Universal Robots PolyScope program: straight floor demo.urp

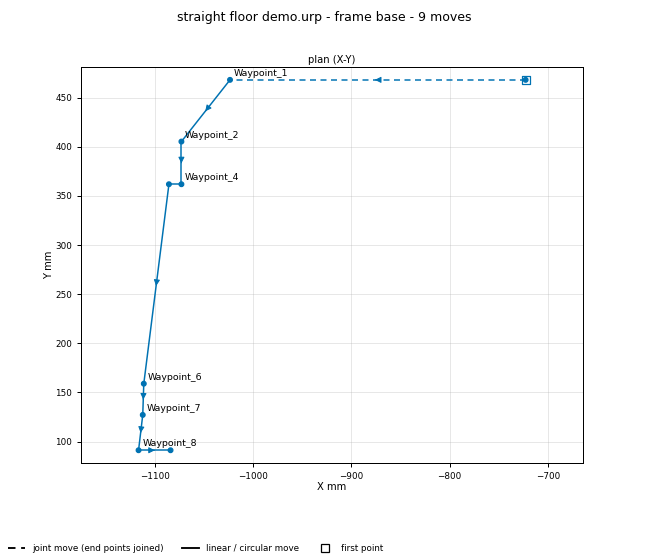
[picture p0: tool path of straight floor demo.urp in frame base, 9 of 9 moves have a stored position in this frame; points joined in program order, loops and branches not executed]
Program straight floor demo (installation=default directory=/programs createdIn=5.21.3 lastSavedIn=5.21.3 robotSerialNumber=20246801938)
Calibrated DH parameters: a=[-0.000071, -0.790281, -0.600694, 0.000061, -0.000039, 0]; d=[0.236272, 604.465945, 132.116513, -736.382239, 0.159268, 0.154005]; alpha=[1.570254, -0.000567, 0.000559, 1.571709, -1.56999, 0]; deltaTheta=[0, -0.409357, 7.293326, -0.600784, -0.000001, -0.000001]
InitVariablesNode
Robot Program (runOnlyOnce=false)
  Folder Folder1
    SuppressedNode
      MoveJ speed 60 deg/s, acceleration 80 deg/s^2 (useActiveTCP=true optimoveEnabled=false optiMoveSpeed=0.3 optiMoveAcceleration=0.09) feature=Base
        Waypoint oldhome: TCP in base x=397.354 y=356.263 z=319.809 mm, rx=2.3163 ry=2.0576 rz=0.0741 rad; joints [-198.308, -118.162, 133.452, -12.561, -11.517, -6.326] deg; TCP offset x=-9.5 y=-328 z=105.73 mm, rx=1.2092 ry=-1.2092 rz=1.2092 rad
    MoveJ speed 60 deg/s, acceleration 80 deg/s^2 (useActiveTCP=true optimoveEnabled=false optiMoveSpeed=0.3 optiMoveAcceleration=0.09) feature=Base
      Waypoint Waypoint_3: TCP in base x=-722.694 y=468.114 z=-58.679 mm, rx=-2.1116 ry=0.3311 rz=2.0412 rad; joints [-64.053, -54.316, 154.48, -187.789, -90.798, 312.597] deg
      Waypoint Waypoint_1: TCP in base x=-1023.509 y=468.114 z=-58.679 mm, rx=-2.1116 ry=0.3311 rz=2.0412 rad; joints [-42.99, -54.355, 134.192, -167.351, -89.902, 333.647] deg
    MoveL speed 20 mm/s, acceleration 1200 mm/s^2 (useActiveTCP=true optimoveEnabled=false optiMoveSpeed=0.3 optiMoveAcceleration=0.09) feature=Base
      Waypoint Waypoint_2: TCP in base x=-1072.965 y=405.321 z=-50.994 mm, rx=2.2388 ry=0.0055 rz=-2.1569 rad; joints [-42.937, -53.961, 129.721, -163.349, -90.663, 315.614] deg
      Waypoint Waypoint_4: TCP in base x=-1072.965 y=361.906 z=-50.994 mm, rx=2.2388 ry=0.0055 rz=-2.1569 rad; joints [-40.714, -54.402, 131.441, -164.605, -90.572, 317.835] deg
      Waypoint Waypoint_5: TCP in base x=-1085.671 y=361.906 z=-50.994 mm, rx=-2.2075 ry=0.1584 rz=2.13 rad; joints [-37.594, -54.591, 132.165, -165.084, -90.081, 329.433] deg
      Waypoint Waypoint_6: TCP in base x=-1111.256 y=158.94 z=-50.994 mm, rx=-2.2075 ry=0.1584 rz=2.13 rad; joints [-24.094, -55.21, 134.996, -167.356, -89.511, 342.92] deg
      Waypoint Waypoint_7: TCP in base x=-1112.305 y=127.176 z=-50.994 mm, rx=2.2506 ry=-0.0217 rz=-2.1687 rad; joints [-24.593, -55.191, 134.842, -167.171, -89.831, 335.324] deg
      Waypoint Waypoint_8: TCP in base x=-1116.578 y=91.213 z=-50.994 mm, rx=2.2506 ry=-0.0217 rz=-2.1687 rad; joints [-22.045, -55.211, 134.953, -167.274, -89.723, 337.87] deg
      Waypoint Waypoint_9: TCP in base x=-1084.025 y=91.213 z=-50.994 mm, rx=2.2506 ry=-0.0217 rz=-2.1687 rad; joints [-22.979, -55.724, 137.618, -169.421, -89.763, 336.936] deg
